{attribute 'qualified_only'}
{attribute 'strict'}
TYPE
    eTcoSmartFunctionKitParticipant :
    (
        WebInterface := 1,
        Fieldbus := 2,
        PhysicalInputsOutputs := 3
    );
END_TYPE

(* stored: Version 1.1.0.1
   DUT eTcoSmartFunctionKitParticipant: Id {2c7c48de-6ab2-40ac-9be2-4f4c489b1dda} *)
